{attribute 'qualified_only'}
{attribute 'strict'}
{attribute 'to_string'}
TYPE E_HomingModes :
(
	Off,	
	MainTest,
	JibTest,
	WinchTest,
	DualTest
);
END_TYPE

(* stored: Version 1.1.0.1
   DUT E_HomingModes: Id {bedadae5-3914-4e8f-8c1f-b0650a0257ff} *)
